FUNCTION_BLOCK PnpXYCalculator (* Basic Function Block Type *)
  (* Standard: 61499-2 *)
  (* Version 0.0, 2/7/2012, XPMUser, nxtControl GmbH, Template *)
  PACKAGE Main;
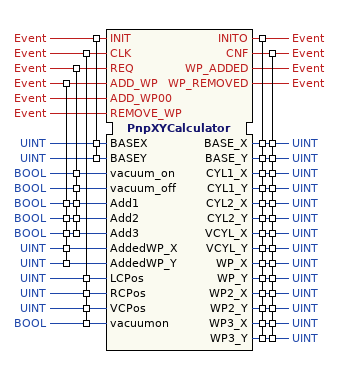
  EVENT_INPUT
    INIT WITH BASEX, BASEY; (* Initialization Request *)
    CLK WITH LCPos, RCPos, VCPos, vacuumon; (* Clock *)
    REQ WITH vacuum_on, vacuum_off, Add1, Add2, Add3;
    ADD_WP WITH Add1, Add2, Add3, AddedWP_X, AddedWP_Y;
    ADD_WP00;
    REMOVE_WP;
  END_EVENT
  EVENT_OUTPUT
    INITO WITH CYL1_X, CYL1_Y, BASE_Y, BASE_X, CYL2_X, CYL2_Y, VCYL_X, VCYL_Y, WP_X, WP_Y, WP2_X, WP2_Y, WP3_X, WP3_Y; (* Initialization Confirm *)
    CNF WITH CYL1_X, CYL1_Y, BASE_Y, BASE_X, CYL2_X, CYL2_Y, VCYL_X, VCYL_Y, WP_X, WP_Y, WP2_X, WP2_Y, WP3_X, WP3_Y;
    WP_ADDED;
    WP_REMOVED;
  END_EVENT
  VAR_INPUT
    BASEX : UINT;
    BASEY : UINT;
    vacuum_on : BOOL;
    vacuum_off : BOOL;
    Add1 : BOOL;
    Add2 : BOOL;
    Add3 : BOOL;
    AddedWP_X : UINT;
    AddedWP_Y : UINT;
    LCPos : UINT;
    RCPos : UINT;
    VCPos : UINT;
    vacuumon : BOOL;
  END_VAR
  VAR_OUTPUT
    BASE_X : UINT; (* Response Data from Socket *)
    BASE_Y : UINT; (* Response Data from Socket *)
    CYL1_X : UINT; (* Response Data from Socket *)
    CYL1_Y : UINT; (* Response Data from Socket *)
    CYL2_X : UINT; (* Response Data from Socket *)
    CYL2_Y : UINT; (* Response Data from Socket *)
    VCYL_X : UINT; (* Response Data from Socket *)
    VCYL_Y : UINT; (* Response Data from Socket *)
    WP_X : UINT; (* Response Data from Socket *)
    WP_Y : UINT; (* Response Data from Socket *)
    WP2_X : UINT; (* Response Data from Socket *)
    WP2_Y : UINT; (* Response Data from Socket *)
    WP3_X : UINT; (* Response Data from Socket *)
    WP3_Y : UINT; (* Response Data from Socket *)
  END_VAR
  VAR
    cyl1x : UINT;
    cyl2x : UINT;
    vcyly : UINT;
    wpx : UINT;
    wpy : UINT;
    wp2x : UINT;
    wp2y : UINT;
    wp3x : UINT;
    wp3y : UINT;
    slider1 : BOOL;
    slider2 : BOOL;
    slider3 : BOOL;
    wpon : BOOL;
    wp2on : BOOL;
    wp3on : BOOL;
  END_VAR
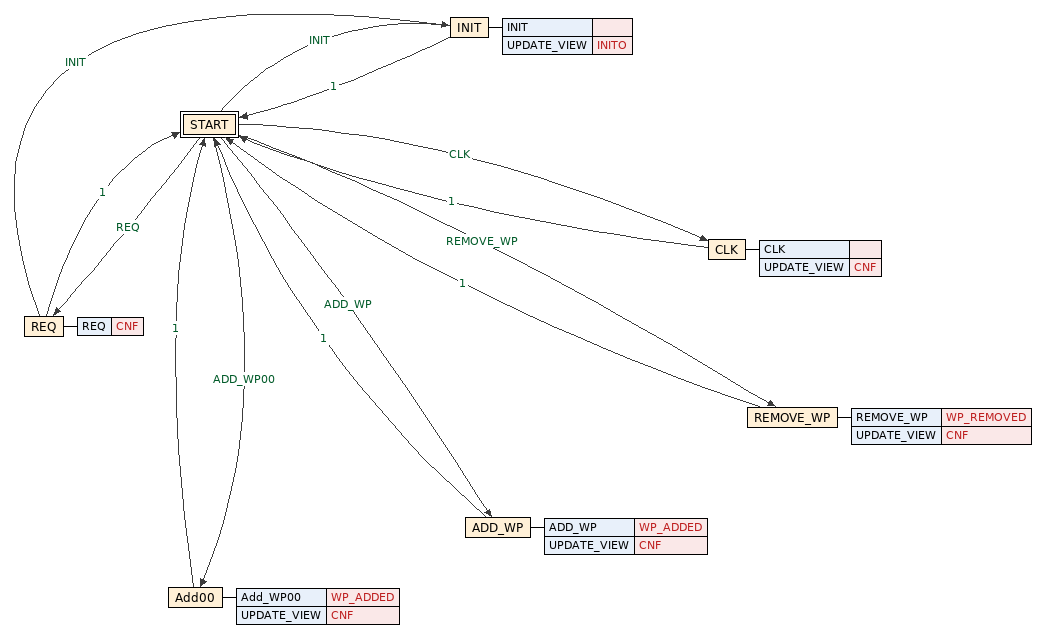
  EC_STATES
    START; (* Initial State *)
    INIT : INIT, UPDATE_VIEW -> INITO; (* Initialization *)
    REQ : REQ -> CNF; (* Normal execution *)
    CLK : CLK, UPDATE_VIEW -> CNF;
    ADD_WP : ADD_WP -> WP_ADDED, UPDATE_VIEW -> CNF;
    REMOVE_WP : REMOVE_WP -> WP_REMOVED, UPDATE_VIEW -> CNF;
    Add00 : Add_WP00 -> WP_ADDED, UPDATE_VIEW -> CNF;
  END_STATES
  EC_TRANSITIONS
    START TO INIT := INIT;
    INIT TO START := 1;
    START TO REQ := REQ;
    REQ TO START := 1;
    START TO CLK := CLK;
    CLK TO START := 1;
    START TO ADD_WP := ADD_WP;
    ADD_WP TO START := 1;
    START TO REMOVE_WP := REMOVE_WP;
    REMOVE_WP TO START := 1;
    START TO Add00 := ADD_WP00;
    Add00 TO START := 1;
    REQ TO INIT := INIT;
  END_TRANSITIONS
  ALGORITHM INIT IN ST: (* Initialization algorithm *)
INIT:=FALSE;
wpx := 6000;
wpy := 6000;
wp2x := 6000;
wp2y := 6000;
wp3x := 6000;
wp3y := 6000;
wpon := FALSE;
wp2on := FALSE;
wp3on := FALSE;

cyl1x := 0;
cyl2x := 0;
vcyly := 0;
slider1 := FALSE;
slider2 := FALSE;
slider3 := FALSE;

BASE_X := BASEX ;
BASE_Y := BASEY ;
CYL1_Y := BASEY ;
CYL2_Y := BASEY +12;
  END_ALGORITHM
  ALGORITHM REQ IN ST: (* Normally executed algorithm *)

  END_ALGORITHM
  ALGORITHM CLK IN ST:
VAR
cyl1_length:INT;
cyl2_length:INT;
vcyl_length:INT;

vacuumx:UINT;
vacuumy:UINT;
dx:UINT;
dy:UINT;
dx2:UINT;
dy2:UINT;
dx3:UINT;
dy3:UINT;

END_VAR
cyl1_length := 75;
cyl2_length := 150;
vcyl_length := 75;

(* horizontal cylinder 1 *)
cyl1x := LCPos;

(* horizontal cylinder 2  *)
cyl2x := RCPos;

(* vertical cylinder  *)
vcyly := VCPos;

IF wpx <= 10 AND wpy >= 185 THEN
    slider1 := TRUE;
ELSE
    slider1 := FALSE;
END_IF;

IF wp2x <= 10 AND wp2y >= 185 THEN
    slider2 := TRUE;
ELSE
    slider2 := FALSE;
END_IF;

IF wp3x <= 10 AND wp3y >= 185 THEN
    slider3 := TRUE;
ELSE
    slider3 := FALSE;
END_IF;

IF vacuumon = TRUE THEN
    vacuumx := cyl1x + cyl2x;
    vacuumy := vcyly + 115;
    dx := ABS(wpx - vacuumx);
    dy := ABS(wpy - vacuumy);
    dx2 := ABS(wp2x - vacuumx);
    dy2 := ABS(wp2y - vacuumy);
    dx3 := ABS(wp3x - vacuumx);
    dy3 := ABS(wp3y - vacuumy);

    IF  dx < 17 AND dy < 7 AND wp2on = FALSE AND wp3on = FALSE THEN
        wpon := TRUE;
    END_IF;

    IF dx2 < 17 AND dy2 < 7 AND wpon = FALSE AND wp3on = FALSE THEN
        wp2on := TRUE;
    END_IF;

    IF dx3 < 17 AND dy3 < 7 AND wp2on = FALSE AND wpon = FALSE THEN
        wp3on := TRUE;
    END_IF;
ELSE
    wpon := FALSE;
    wp2on := FALSE;
    wp3on := FALSE;
END_IF;
  END_ALGORITHM
  ALGORITHM UPDATE_VIEW IN ST:
VAR
bx:UINT;
byy:UINT;
END_VAR
bx := BASEX;
byy := BASEY;

CYL1_X  := bx + 22 + cyl1x ;
CYL2_X  := bx + 116 + cyl1x + cyl2x ;
VCYL_X  := bx + 305 + cyl1x + cyl2x ;
VCYL_Y  := byy + vcyly + 15;

IF wpon = TRUE  THEN
    wpx  := cyl1x + cyl2x ;
    wpy  := vcyly + 115;
ELSIF slider1 = TRUE THEN
    wpy  := wpy + 1;
ELSE
    wpy  := 190;
END_IF;

IF wp2on = TRUE THEN
    wp2x  := cyl1x + cyl2x ;
    wp2y  := vcyly + 115;
ELSIF slider2 = TRUE THEN
    wp2y  := wp2y + 1;
ELSE
    wp2y  := 190;
END_IF;

IF wp3on = TRUE THEN
    wp3x  := cyl1x + cyl2x ;
    wp3y  := vcyly + 115;
ELSIF slider3 =TRUE THEN
    wp3y  := wp3y + 1;
ELSE
    wp3y  := 190;
END_IF;

WP_X  := bx + 300 + wpx ;
WP_Y  := byy + wpy ;
WP2_X := bx + 300 + wp2x ;
WP2_Y := byy + wp2y ;
WP3_X := bx + 300 + wp3x ;
WP3_Y := byy + wp3y ;
IF WP_X  = 305 AND WP_Y  >= 330 THEN
    WP_X  := 6000;
    WP_Y  := 6000;
END_IF;
IF WP2_X  = 305 AND WP2_Y  >= 330 THEN
    WP2_X  := 6000;
    WP2_Y  := 6000;
END_IF;
IF WP3_X  = 305 AND WP3_Y  >= 330 THEN
    WP3_X  := 6000;
    WP3_Y  := 6000;
END_IF;
  END_ALGORITHM
  ALGORITHM ADD_WP IN ST:
IF Add1 = TRUE THEN
wpx := 75;
wpy := 215;
wpon := FALSE;
END_IF;
IF Add2 = TRUE THEN
wp2x := 150;
wp2y := 215;
wp2on := FALSE;
END_IF;
IF Add3 = TRUE THEN
wp3x := 225;
wp3y := 215;
wp3on := FALSE;
END_IF;
  END_ALGORITHM
  ALGORITHM REMOVE_WP IN ST:

  END_ALGORITHM
  ALGORITHM Add_WP00 IN ST:

  END_ALGORITHM
END_FUNCTION_BLOCK
